Universal Robots PolyScope program: motor_orient_3.urp

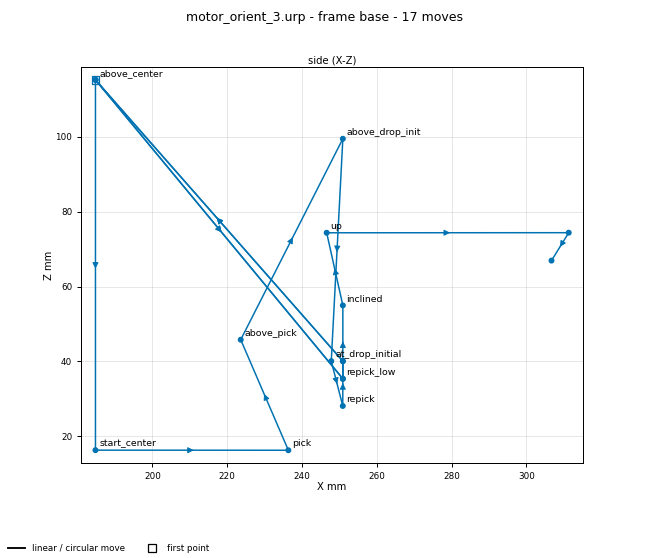
[picture p0: tool path of motor_orient_3.urp in frame base, 17 of 18 moves have a stored position in this frame; points joined in program order, loops and branches not executed]
Program motor_orient_3 (installation=default directory=/programs/wrs2020 createdIn=5.10.0.106288 lastSavedIn=5.10.0.106288 robotSerialNumber=20205500607)
Calibrated DH parameters: a=[0.000096, -0.337, -0.383372, 0.000118, 0.000015, 0]; d=[0.162724, 79.377998, -95.545185, 16.300583, 0.099689, 0.099499]; alpha=[1.569249, 0.003272, 0.005201, 1.570041, -1.570219, 0]; deltaTheta=[0, 0.65664, 5.410619, 0.215927, -0.000001, 0]
Robot Program (runOnlyOnce=true)
  MoveJ speed 180 deg/s, acceleration 120 deg/s^2 (useActiveTCP=false) tcp=gripper_85_tip; feature=Base
    currentpose := get_actual_joint_positions()
    Waypoint Waypoint (Variable): variable=currentpose
  Folder center
    MoveJ speed 180 deg/s, acceleration 120 deg/s^2 (useActiveTCP=true) feature=Base
      Waypoint above_center: TCP in base x=184.767 y=-168.569 z=115.27 mm, rx=-2.2265 ry=2.1698 rz=0.0754 rad; joints [105.603, -125.054, 143.664, -105.259, -89.614, -76.004] deg; TCP offset x=0 y=0 z=165 mm, rx=0 ry=0 rz=0 rad
    MoveL speed 250 mm/s, acceleration 1200 mm/s^2 (useActiveTCP=true) feature=Base
      Waypoint start_center: TCP in base x=184.767 y=-168.568 z=16.246 mm, rx=-2.2265 ry=2.1698 rz=0.0754 rad; joints [105.483, -111.397, 155.293, -130.549, -89.612, -75.992] deg
      MoveDirectionNode (selectedDirection=XPlus toolParams=0.008, 0.01) feature=Base
        Until TOOL_CONTACT_DETECTION (allowActions=false retraction=NONE decelerationAcceleration=3 decelerationAngularAcceleration=34.906585)
      URCap Gripper (Robotiq_Grippers, Robotiq Inc.) dataModel(position=0.0, force=100.0, speed=100.0, positionInDouble=0.0, forceInDouble=100.0, speedInDouble=100.0, slaveIds=[9], blocking=false)
  Folder pick
    SuppressedNode
      URCap Gripper (Robotiq_Grippers, Robotiq Inc.) dataModel(position=0.0, force=100.0, speed=100.0, positionInDouble=0.0, forceInDouble=100.0, speedInDouble=100.0, slaveIds=[9], blocking=false)
    SuppressedNode
      MoveJ speed 60 deg/s, acceleration 80 deg/s^2 (useActiveTCP=true) feature=Base
        Waypoint above_pick: TCP in base x=118.06 y=-247.674 z=105.282 mm, rx=-0.1162 ry=3.083 rz=0.0206 rad; joints [83.323, -121.678, 144.556, -111.588, -86.705, -11.125] deg
    MoveL speed 500 mm/s, acceleration 800 mm/s^2 (useActiveTCP=true) feature=Base
      Waypoint pick: TCP in base x=236.349 y=-168.533 z=16.223 mm, rx=-2.2264 ry=2.1698 rz=0.0755 rad; joints [116.573, -102.278, 150.321, -134.785, -88.96, -64.891] deg
      URCap Gripper (Robotiq_Grippers, Robotiq Inc.) dataModel(position=100.0, force=100.0, speed=100.0, positionInDouble=100.0, forceInDouble=100.0, speedInDouble=100.0, slaveIds=[9], blocking=true)
      Waypoint above_pick: motionParameters(blendRadius=0.009); TCP in base x=223.61 y=-168.561 z=45.782 mm, rx=-2.2266 ry=2.1698 rz=0.0754 rad; joints [114.122, -109.864, 148.803, -125.653, -89.103, -67.391] deg
  Folder 10 drops
    MoveL speed 800 mm/s, acceleration 800 mm/s^2 (useActiveTCP=true) feature=Base
      Waypoint above_drop_init: motionParameters(blendRadius=0.05); TCP in base x=250.92 y=-170.231 z=99.518 mm, rx=-2.207 ry=2.1484 rz=-0.0127 rad; joints [116.629, -114.877, 142.708, -117.082, -86.275, -64.998] deg
      Waypoint at_drop_initial: TCP in base x=247.821 y=-170.422 z=40.046 mm, rx=-2.2069 ry=2.1485 rz=-0.0127 rad; joints [115.955, -107.181, 149.284, -131.319, -86.287, -65.596] deg
      URCap Gripper (Robotiq_Grippers, Robotiq Inc.) dataModel(position=25.88235294117647, force=100.0, speed=100.0, positionInDouble=25.88235294117647, forceInDouble=100.0, speedInDouble=100.0, slaveIds=[9], blocking=true)
      Loop Counting (count=3) loopVariable(name=Loop_1)
        Waypoint repick: TCP in base x=250.899 y=-170.231 z=28.067 mm, rx=-2.2069 ry=2.1485 rz=-0.0126 rad; joints [116.558, -104.445, 150.108, -134.913, -86.284, -64.971] deg
        URCap Gripper (Robotiq_Grippers, Robotiq Inc.) dataModel(position=100.0, force=100.0, speed=100.0, positionInDouble=100.0, forceInDouble=100.0, speedInDouble=100.0, slaveIds=[9], blocking=true)
        Waypoint redrop: TCP in base x=250.921 y=-170.242 z=40.048 mm, rx=-2.2069 ry=2.1485 rz=-0.0127 rad; joints [116.571, -106.658, 148.996, -131.592, -86.279, -64.975] deg
        If rq_current_pos_mm() < 10
          Waypoint above_center: TCP in base x=184.767 y=-168.569 z=115.27 mm, rx=-2.2265 ry=2.1698 rz=0.0754 rad; joints [105.603, -125.054, 143.664, -105.259, -89.614, -76.004] deg
          Halt
        URCap Gripper (Robotiq_Grippers, Robotiq Inc.) dataModel(blocking=true, slaveIds=[9], speedInDouble=100.0, forceInDouble=100.0, positionInDouble=25.88235294117647, speed=100.0, force=100.0, position=25.88235294117647)
      Loop Counting (count=3) loopVariable(name=Loop_2)
        Waypoint repick_low: TCP in base x=250.923 y=-170.228 z=35.335 mm, rx=-2.2069 ry=2.1485 rz=-0.0127 rad; joints [116.565, -105.813, 149.441, -132.88, -86.276, -64.974] deg
        URCap Gripper (Robotiq_Grippers, Robotiq Inc.) dataModel(position=100.0, force=100.0, speed=100.0, positionInDouble=100.0, forceInDouble=100.0, speedInDouble=100.0, slaveIds=[9], blocking=true)
        Waypoint redrop: TCP in base x=250.921 y=-170.242 z=40.048 mm, rx=-2.2069 ry=2.1485 rz=-0.0127 rad; joints [116.571, -106.658, 148.996, -131.592, -86.279, -64.975] deg
        If rq_current_pos_mm() < 10
          Waypoint above_center: TCP in base x=184.767 y=-168.569 z=115.27 mm, rx=-2.2265 ry=2.1698 rz=0.0754 rad; joints [105.603, -125.054, 143.664, -105.259, -89.614, -76.004] deg
          Halt
        SuppressedNode
          URCap Gripper (Robotiq_Grippers, Robotiq Inc.) dataModel(position=25.88235294117647, force=100.0, speed=100.0, positionInDouble=25.88235294117647, forceInDouble=100.0, speedInDouble=100.0, slaveIds=[9], blocking=true)
        URCap Gripper (Robotiq_Grippers, Robotiq Inc.) dataModel(position=0.0, force=0.0, speed=0.0, positionInDouble=0.0, forceInDouble=0.0, speedInDouble=0.0, slaveIds=[9], blocking=true)
  Folder place
    MoveL speed 250 mm/s, acceleration 1200 mm/s^2 (useActiveTCP=true) feature=Base
      Waypoint pick2: TCP in base x=250.923 y=-170.228 z=35.335 mm, rx=-2.2069 ry=2.1485 rz=-0.0127 rad; joints [116.565, -105.813, 149.441, -132.88, -86.276, -64.974] deg
      URCap Gripper (Robotiq_Grippers, Robotiq Inc.) dataModel(position=0.0, force=0.0, speed=0.0, positionInDouble=0.0, forceInDouble=0.0, speedInDouble=0.0, slaveIds=[9], blocking=true)
      Waypoint inclined: TCP in base x=250.917 y=-170.201 z=54.957 mm, rx=2.2249 ry=-2.1708 rz=-0.118 rad; joints [122.621, -104.551, 143.845, -125.427, -92.46, -58.708] deg
      MoveDirectionNode (selectedDirection=XPlus toolParams=0.004, 0.01)
        Until TOOL_CONTACT_DETECTION (allowActions=false retraction=0.01 decelerationAcceleration=3 decelerationAngularAcceleration=34.906585)
      Waypoint up: TCP in base x=246.593 y=-170.172 z=74.376 mm, rx=2.2249 ry=-2.1708 rz=-0.118 rad; joints [121.927, -107.874, 142.374, -120.664, -92.506, -59.427] deg
      Waypoint forward: TCP in base x=311.323 y=-170.194 z=74.399 mm, rx=2.2248 ry=-2.1708 rz=-0.1179 rad; joints [131.177, -97.986, 135.309, -123.097, -91.837, -50.168] deg
      Waypoint place: motionParameters(jointSpeed=1.047198 jointAcceleration=1.396263 cartesianSpeed=0.02 cartesianAcceleration=1.2); TCP in base x=306.715 y=-169.627 z=66.937 mm, rx=2.2249 ry=-2.1707 rz=-0.1179 rad; joints [130.662, -97.796, 136.545, -124.543, -91.876, -50.678] deg
      URCap Gripper (Robotiq_Grippers, Robotiq Inc.) dataModel(position=1.1764705882352942, force=0.0, speed=0.0, positionInDouble=1.1764705882352942, forceInDouble=0.0, speedInDouble=0.0, slaveIds=[9], blocking=true)
  SuppressedNode
    Folder touch
      MoveL speed 250 mm/s, acceleration 1200 mm/s^2 (useActiveTCP=true) feature=Base
        Waypoint touch: TCP in base x=350.448 y=-169.715 z=63.797 mm, rx=-2.1526 ry=2.2403 rz=-0.0049 rad; joints [132.881, -94.454, 135.596, -131.257, -87.731, -44.801] deg
        URCap Gripper (Robotiq_Grippers, Robotiq Inc.) dataModel(position=100.0, force=100.0, speed=100.0, positionInDouble=100.0, forceInDouble=100.0, speedInDouble=100.0, slaveIds=[9], blocking=true)
        URCap Gripper (Robotiq_Grippers, Robotiq Inc.) dataModel(position=0.0, force=100.0, speed=100.0, positionInDouble=0.0, forceInDouble=100.0, speedInDouble=100.0, slaveIds=[9], blocking=true)
